FUNCTION_BLOCK FB_ImmersionHeater
VAR_INPUT
END_VAR
VAR_OUTPUT
END_VAR
VAR
END_VAR

END_FUNCTION_BLOCK

(* stored: Version 1.1.0.1, ProductVersion 3.1.4024.10
   POU FB_ImmersionHeater: Id {2de23c48-52f9-4c7c-a711-bae727744ee8}, SpecialFunc None *)
